TEXTLIST Alarm_list
  0 = 'No Alarm'
  1 = 'Emergency stop Pressed'
  2 = 'Home action Interlock error-CC1 \tClamp'
  3 = 'Home action timeout error-CC1 \tClamp'
  4 = 'Work action Interlock error-CC1 \tClamp'
  5 = 'Work action timeout error-CC1 \tClamp'
  6 = 'Home action Interlock error-CC2 \tClamp'
  7 = 'Home action timeout error-CC2\t Clamp'
  8 = 'Work action Interlock error-CC2 \tClamp'
  9 = 'Work action timeout error-CC2 \tClamp'
  10 = 'Home action Interlock error-CC3 \tClamp'
  11 = 'Home action timeout error-CC3\t Clamp'
  12 = 'Work action Interlock error-CC3 \tClamp'
  13 = 'Work action timeout error-CC3 \tClamp'
  14 = 'Home action Interlock error-CC4 \tClamp'
  15 = 'Home action timeout error-CC4\t Clamp'
  16 = 'Work action Interlock error-CC4 \tClamp'
  17 = 'Work action timeout error-CC4 \tClamp'
  18 = 'Home action Interlock error-CC5 \tClamp'
  19 = 'Home action timeout error-CC5\t Clamp'
  20 = 'Work action Interlock error-CC5 \tClamp'
  21 = 'Work action timeout error-CC5 \tClamp'
  22 = 'Home action Interlock error-CC6 \tClamp'
  23 = 'Home action timeout error-CC6\t Clamp'
  24 = 'Work action Interlock error-CC6 \tClamp'
  25 = 'Work action timeout error-CC6 \tClamp'
   = ''
END_TEXTLIST

(* stored: Version 1.1.0.1, ProductVersion 3.1.4024.16
   TextList Alarm_list: Id {5cb2479c-7173-489f-89c9-4400f09acf02} *)
